{attribute 'qualified_only'}
VAR_GLOBAL CONSTANT
	COMMAND_BUFFER_SIZE :UDINT := 63; // Queue size for database insert command.
END_VAR

(* stored: Version 1.1.0.1, ProductVersion 3.1.4024.12
   GVL LibraryParameter: Id {56321c42-7c93-46e8-98ed-6ddc16ce704e}, ParameterList True *)
